TYPE STRUCT_AxisExtendedCompound :
STRUCT
	
	Ref:		AXIS_REF;
	Crtl:		ExtendedAxisTyp;
	
END_STRUCT
END_TYPE

(* stored: Version 1.1.0.1, ProductVersion 3.1.4024.3
   DUT STRUCT_AxisExtendedCompound: Id {2422cd1b-d22b-0b97-04d2-73ccf3c439a0} *)
